DATA_BLOCK "ST10_FB_S7connect_IDB"
VAR
  Always_On : Bool;
  Status_Get : Array[1..6] of Struct;
  Status_Put : Array[1..6] of Struct;
  GET_Instance1 : GET;
  GET_Instance2 : GET;
  PUT_Instance1 : PUT;
  PUT_Instance2 : PUT;
  PLs : Array[1..6] of Bool;
  TON : Array[1..5] of TON_TIME;
  NextStation_OffLine : Bool;
END_VAR
BEGIN
END_DATA_BLOCK
